FUNCTION_BLOCK Turntable
VAR_INPUT



END_VAR
VAR_OUTPUT

	bTurn 		: BOOL;
	bRollPlus	: BOOL;
	bRollMinus 	: BOOL;
	bFrontLimit : BOOL;
	bBackLimit	: BOOL;
	
END_VAR
VAR

	fbFrontLimit : Sensor;
	fbBackLimit : Sensor;
	
	fbTurn : BoolOut;
	fbRollPlus : BoolOut;
	fbRollMinus : BoolOut;
	
END_VAR

fbFrontLimit();
fbBackLimit();

bTurn := fbTurn.getValue;
bRollPlus := fbRollPlus.getValue;
bRollMinus := fbRollMinus.getValue;
bFrontLimit := fbFrontLimit.bSignal;
bBackLimit	:= fbBackLimit.bSignal;

METHOD RollMinus : BOOL
VAR_INPUT
END_VAR
fbRollMinus.setValue := TRUE;
fbRollPlus.setValue := FALSE;
END_METHOD

METHOD RollPlus : BOOL
VAR_INPUT
END_VAR
fbRollPlus.setValue := TRUE;
fbRollMinus.setValue := FALSE;
END_METHOD

METHOD StopRolling : BOOL
VAR_INPUT
END_VAR
fbRollMinus.setValue := FALSE;
fbRollPlus.setValue := FALSE;
END_METHOD

METHOD Turn : BOOL
VAR_INPUT
END_VAR
fbTurn.setValue := TRUE;
END_METHOD

METHOD Unturn : BOOL
VAR_INPUT
END_VAR
fbTurn.setValue := FALSE;
END_METHOD

END_FUNCTION_BLOCK

(* stored: Version 1.1.0.1, ProductVersion 3.1.4024.2
   POU Turntable: Id {d4c6f4bb-289d-40ee-a543-6dd70783c627}, SpecialFunc None
   Method RollMinus: Id {6cce44bf-5b3c-4c9b-9d87-b3e968d8e2cd}
   Method RollPlus: Id {06d4d60b-912a-4be3-a693-5f84ed719d3a}
   Method StopRolling: Id {db8d8c41-df94-4d38-8c5e-204aabd95a55}
   Method Turn: Id {e767dad2-b25c-4cbc-87f3-f7bd7f84290a}
   Method Unturn: Id {1e1fa2db-0d4e-4205-a5ad-f257eb1d93eb} *)
